// TIA Portal V19 export
TYPE "typeU2Em1Para"
// stored: Access Published
   STRUCT
      cm1Vfd205 : "typeVfdInterface";
   END_STRUCT;
END_TYPE
